// Mitsubishi GX Works2 project: 2   PLC: FX3U/FX3UC

// task Task_01 (event TRUE, interval 0, priority 31): POU_01

PROGRAM POU_01
VAR
  wstep : INT;
  R_TRIG_THRY_1 : R_TRIG;
  R_TRIG_THRY_2 : R_TRIG;
  R_TRIG_THRY_3 : R_TRIG;
  TON_SYNC : TON;
END_VAR
M99 := 
Y1 AND Y2 AND Y3 AND Y4 AND
Y0 AND
Y11 AND Y12 AND Y13 AND Y14 AND

X1 AND X2 AND X3 AND X4 AND X5 AND
X0 AND
X11 AND X12 AND
X15 AND X16 AND X17 AND 
X6 AND X7 AND X10 AND X14;

(*PB1- X1*)						(*PL1 - Y1*)
(*PB2 - X2*)						(*PL2 - Y2*)
(*PB3 - X3*)						(*PL3 - Y3*)
(*PB4  - X4*)						(*PL4 - Y4*)
(*PB5 - X5*)						(*BZ - Y0*)
(*EMS NC - X0*)				(*MC1 - Y11*)
(*COS 1 - X11*)				(*MC2 - Y12*)
(*COS 2 - X12*)				(*MC3 - Y13*)
(*TH-RY 1 NC - X15*)		(*MC4 - Y14*)
(*TH-RY 2 NC - X16*)
(*TH-RY 3 NC - X17*)
(*MC1 NO - X6*)			
(*MC2 NO - X7*)
(*MC3 NO - X10*)
(*MC4 NO - X14*)

IF M8002 THEN
	wstep := 0;
END_IF;

IF wstep <> 50 THEN (*MC無法同步*)
	(*EMS*)
	IF NOT X0 THEN 
		wstep := 0;
	END_IF;
	
	(*過載警示*)
	IF NOT (X15 AND X16 AND X17) THEN
		Y4 := M8013 OR ((NOT X11) AND X12);
		Y0 := NOT M8013 AND (X11 AND (NOT X12)); 
	ELSE
		RST(TRUE, Y4);
		RST(TRUE, Y0);
	END_IF;
	
	(*TH-RY 過載控制*)
	IF NOT X17 THEN
		ZRST(TRUE, Y11, Y14);
		ZRST(TRUE, Y1, Y3);
	END_IF;
	
	IF NOT X16 THEN
		ZRST(TRUE, Y11, Y12);
		ZRST(TRUE, Y1, Y2);
	END_IF;
	
	IF NOT X15 THEN
		RST(TRUE, Y11);	
		RST(TRUE, Y1);	
	END_IF;
END_IF;

(*MC無法同步*)
TON_SYNC(IN := (X6 XOR Y11) OR (X7 XOR Y12) OR (X10 XOR Y13) OR (X14 XOR Y14), PT := T#2s);
IF TON_SYNC.Q THEN
	wstep := 50;
END_IF;

CASE wstep OF 
	0: (*正常情況*)
		ZRST(TRUE , Y1, Y3);
		ZRST(TRUE , Y5, Y17);
		ZRST(TRUE , TC0, TC200);
		IF X0 AND X17 THEN (*COS轉到 1 ; EMS為無按下 ; 無過載*)
			IF X3 THEN
				wstep := 20;
			END_IF;
			IF X2 THEN
				wstep := 30;
			END_IF;
		END_IF;
		
	20: (*手動*)
		IF NOT X17 THEN (*過載則返回*)
			wstep := 0;
		END_IF;
		SET(TRUE, Y13);
		SET(TRUE, Y14);
		SET(TRUE, Y3);
		IF X4 AND X16 THEN
			wstep := 21;
		END_IF;
	21:
		IF NOT (X17 AND X16) THEN (*過載則返回*)
			wstep := 20;
		END_IF;
		SET(TRUE, Y12);
		SET(TRUE, Y2);
		IF X5 AND X15 THEN
			wstep := 22;
		END_IF;
	22:
		IF NOT (X17 AND X16 AND X15) THEN (*過載則返回*)
			wstep := 21;
		END_IF;
		SET(TRUE, Y11);
		SET(TRUE, Y1);
		IF X1 THEN
			wstep := 40;
		END_IF;
	
	30: (*自動*)
		IF NOT X17 THEN (*過載則返回*)
			wstep := 21;
		END_IF;
		SET(TRUE, Y13);
		SET(TRUE, Y14);
		Y3 := M8013;
		OUT_T(TRUE, TC0, 50);
		IF TS0 THEN
			wstep := 31;
		END_IF;
	31:
		IF NOT (X17 AND X16) THEN (*過載則返回*)
			wstep := 21;
		END_IF;
		SET(TRUE, Y3);
		SET(TRUE, Y12);
		Y2 := M8013;
		OUT_T(TRUE, TC1, 100);
		IF TS1 THEN
			wstep := 32;
		END_IF;
	32:
		IF NOT (X17 AND X16 AND X15) THEN (*過載則返回*)
			wstep := 21;
		END_IF;
		SET(TRUE, Y2);
		SET(TRUE, Y11);
		SET(TRUE, Y1);
		IF X1 THEN
			ZRST(TRUE, TC0, TC1);
			wstep := 40;
		END_IF;
		
	40: (*關機*)
		RST(TRUE, Y11);
		RST(TRUE, Y1);
		Y2 := M8013;
		OUT_T(TRUE, TC0, 50);
		IF TS0 THEN
			wstep := 41;
		END_IF;
	41:
		RST(TRUE, Y12);
		RST(TRUE, Y2);
		Y3 := M8013;
		OUT_T(TRUE, TC1, 100);
		IF TS1 THEN
			wstep := 0;
		END_IF;
		
	50:
		ZRST(TRUE, Y0, Y17);
END_CASE;
END_PROGRAM
